Yaskawa INFORM job: R1_W27-A5(90,0)OK-KM.JBI

/JOB
//NAME R1_W27-A5(90,0)OK-KM
///FOLDERNAME KRIS-SCIANA
//POS
///NPOS 202,202,0,12,0,0
///TOOL 0
///POSTYPE PULSE
///PULSE
C00000=17399,70332,19465,-6085,71765,84469
C00001=-37728,-26470,-57837,-12171,79874,87707
C00002=-91138,-151926,-106227,-11663,-44198,37632
C00003=-119745,-150224,-99473,-11370,-45552,35827
C00004=-119745,-150224,-99473,27647,23434,35827
C00005=-82911,-32219,-20746,39404,39160,51491
C00006=-76873,-22201,-13846,34402,37292,54508
C00007=-77767,-15549,-470,39111,33772,51878
C00008=-77963,-13883,2721,40331,32997,51211
C00009=-77963,-13524,3630,40708,32708,51011
C00010=-77963,-13883,2721,40331,32997,51211
C00011=-74912,-26998,-14766,34305,34919,54616
C00012=-87425,-26616,-10195,45168,38615,47962
C00013=-86506,-23763,-6209,45546,37441,47802
C00014=-85850,-22824,-4885,45481,36871,47882
C00015=-86506,-23763,-6209,45546,37441,47802
C00016=-88499,-28370,-15308,43879,40777,48661
C00017=-84065,-38855,-25026,49333,30926,46354
C00018=-97660,-56634,-43247,77155,50749,43385
C00019=-97660,-56634,-43247,77155,50749,-23479
C00020=-84258,-2041,-18253,34253,81408,-37843
C00021=-71650,45427,35116,30336,65668,-37926
C00022=-68559,52359,37552,21834,71082,-35585
C00023=-68559,52806,39758,21974,70033,-35786
C00024=-71650,45427,35116,30336,65668,-37926
C00025=-70945,44875,34529,30103,65482,-37681
C00026=-71650,45427,35116,30336,65668,-37926
C00027=-73638,27357,13179,30116,70049,-37523
C00028=-84818,-6426,-32553,25443,106560,-66628
C00029=-82304,-18386,-36135,24935,102238,-66641
C00030=-82304,-18454,-35234,24871,101700,-66756
C00031=-82304,-18386,-36135,24935,102238,-66641
C00032=-81928,-19848,-37209,24925,102044,-66542
C00033=-82304,-18386,-36135,24935,102238,-66641
C00034=-89590,-10771,-36844,25462,108330,-68030
C00035=-79821,25001,-10397,14026,108535,51508
C00036=-75346,31907,-3594,13981,107184,52914
C00037=-69367,42190,15961,2624,107533,53589
C00038=-69672,41458,15193,2593,107639,53485
C00039=-69367,42204,15728,2627,107683,53592
C00040=-69778,41287,13778,2594,108424,53461
C00041=-69778,41233,14455,2587,107981,53452
C00042=-69778,41399,12679,2608,109158,53478
C00043=-75546,31218,-6024,2098,115588,51477
C00044=-89590,-10931,-36200,25384,107896,-68129
C00045=-81318,-17186,-40796,25354,105117,-65637
C00046=-81011,-18361,-41666,25340,104964,-65554
C00047=-81318,-17186,-40796,25354,105117,-65637
C00048=-81318,-16843,-42196,25499,106059,-65424
C00049=-80508,-20067,-43878,25399,105256,-65302
C00050=-80508,-20199,-43312,25343,104878,-65387
C00051=-80508,-20067,-43878,25399,105256,-65302
C00052=-95846,-36703,-51984,36140,101059,-70811
C00053=-102769,-66525,-54062,50542,79902,-82074
C00054=-102006,-66230,-53915,50487,79519,-81882
C00055=-101071,-65850,-53726,50414,79053,-81646
C00056=-102358,-66368,-53984,50514,79697,-81972
C00057=-109446,-45740,-47717,50613,88014,-81159
C00058=-76818,1585,-28485,25537,105673,-88163
C00059=-74377,-650,-29244,25352,104344,-87556
C00060=-73964,-576,-29181,25336,104222,-87428
C00061=-74377,-650,-29244,25352,104344,-87556
C00062=-74377,-197,-30716,25505,105375,-87324
C00063=-73295,556,-29557,25411,104765,-87062
C00064=-73295,319,-28784,25333,104224,-87184
C00065=-73295,556,-29557,25411,104765,-87062
C00066=-75164,936,-29240,25491,105307,-87630
C00067=-75164,673,-28375,25400,104701,-87767
C00068=-73992,-54,-28979,25351,104361,-87410
C00069=-74218,1135,-29725,25504,105397,-87259
C00070=-70279,39917,7631,24946,101471,-86677
C00071=-70279,39773,8340,24894,101006,-86779
C00072=-70279,39917,7631,24946,101471,-86677
C00073=-71244,40896,8655,24982,101636,-86998
C00074=-70901,41500,10265,24911,100916,-87026
C00075=-70430,41573,10341,24887,100771,-86884
C00076=-70902,41494,10304,24893,100890,-87032
C00077=-61413,47913,18827,22376,82611,-84527
C00078=-60983,48200,19135,22272,82457,-84404
C00079=-61413,47913,18827,22376,82611,-84527
C00080=-61413,48031,17812,22351,83248,-84408
C00081=-60688,48267,18121,22175,82995,-84198
C00082=-60688,48184,18825,22194,82554,-84280
C00083=-60688,48216,18544,22185,82728,-84248
C00084=-61554,48611,18972,22401,82900,-84527
C00085=-61554,48574,19313,22409,82686,-84566
C00086=-61046,48574,19311,22284,82551,-84409
C00087=-61144,49040,18429,22280,83303,-84304
C00088=-63518,19819,-3959,31003,65918,-85445
C00089=-64098,13990,-8483,32812,62419,-85700
C00090=-68885,5858,-4837,49954,39982,-79267
C00091=-65088,14401,2351,47338,37926,-77932
C00092=-64176,16514,4289,46758,37375,-77645
C00093=-64374,16048,3860,46884,37498,-77706
C00094=-64374,16332,5960,47994,36717,-78332
C00095=-65291,19511,8504,48605,37238,-78641
C00096=-67140,20670,8164,49136,38778,-78870
C00097=-66295,22610,10004,48674,38233,-78640
C00098=-66438,22276,9687,48752,38326,-78678
C00099=-66438,22593,11839,49879,37554,-79321
C00100=-66183,17456,6587,49121,37801,-78900
C00101=-69997,303,-8544,51199,40225,-79947
C00102=-70090,462,-8411,51396,40399,61925
C00103=-64431,-7994,-19990,55211,47136,55293
C00104=-59732,2731,-7253,54624,43014,55385
C00105=-61112,6047,-4408,55407,43795,54965
C00106=-58127,6230,-5593,41789,36796,53014
C00107=-57063,4244,-3023,44477,29101,47198
C00108=-49270,4507,-14230,7230,38635,77567
C00109=-52170,-21028,-34442,10411,38272,75983
C00110=-53236,-23757,-36400,11576,38221,75401
C00111=-68411,-26721,-55288,29669,69158,-83075
C00112=-64998,-22231,-39429,29595,61484,-83843
C00113=-47332,3156,-26714,14390,83656,-86934
C00114=-13581,-13792,-41839,5505,90345,-85819
C00115=-16349,-25840,-50577,5581,88837,-86870
C00116=-22627,-48080,-64721,6235,84990,-89226
C00117=-44284,-42364,-63168,13491,82223,-86082
C00118=-48658,384,-30330,14766,84654,-87257
C00119=-13581,-13639,-42286,5505,90698,-85803
C00120=-13581,-13792,-41839,5505,90345,-85819
C00121=-42831,1170,-27974,7852,83268,-89098
C00122=-45008,27799,-716,8149,72970,-89221
C00123=-49813,9029,-19459,14067,72438,-89467
C00124=-51221,-59792,-71163,13641,70093,-81113
C00125=-20731,-35064,-57255,13295,95296,-88132
C00126=-10350,-61458,-73206,13150,96697,-81231
C00127=-18568,-72839,-84924,10276,90748,-67361
C00128=-26792,-78269,-88347,11582,91154,33243
C00129=-45042,-56045,-41152,29344,86284,26690
C00130=-29931,-96865,-59275,30269,72400,28931
C00131=-11330,-93733,-53223,18734,61624,35066
C00132=-13142,-100438,-49115,27852,43711,29575
C00133=-45210,-99902,-50498,43944,62722,17519
C00134=-65059,-105763,-56440,35236,62434,-70425
C00135=-52273,-68840,-35855,24782,78790,-57994
C00136=-44191,-94324,-39451,26680,66575,-57785
C00137=-27622,-61862,-26687,25544,69625,-50822
C00138=-34229,-65282,-33006,25339,73525,-52443
C00139=-29998,-45056,-20412,5383,50998,-19853
C00140=-26959,-13487,10958,4231,47743,-18704
C00141=-30725,7190,27774,5945,48250,-20332
C00142=-26399,12630,34412,-7054,43656,-17025
C00143=-25910,12791,35044,-8483,42971,-16590
C00144=-25523,14356,36662,-10737,43316,-14707
C00145=-25240,1993,23649,-9803,41847,-14580
C00146=-22231,-26812,-1283,-11497,42767,-13220
C00147=-78144,-22833,-14293,20182,52194,33247
C00148=-71297,46898,32867,2677,100084,44239
C00149=-55011,25089,17646,-3023,105619,49711
C00150=-60812,41513,34008,-4227,103729,47709
C00151=-58235,32548,20742,-3759,107403,48505
C00152=-79593,-22722,-23344,19568,57852,33734
C00153=-78528,-18616,-11242,20296,52560,33151
C00154=-78932,-16743,-10167,20417,52946,33052
C00155=-78544,-16737,-8595,20480,51941,33014
C00156=-77955,-18452,-11115,20012,52425,33380
C00157=-78575,-16130,-9486,20269,52757,33170
C00158=-76564,-15411,-8500,18566,50879,33728
C00159=-75844,-13833,-7410,18312,50740,34021
C00160=-76952,-15561,-8970,19469,52340,33810
C00161=-76532,-19770,-12086,19320,52008,33932
C00162=-90733,-10813,-5342,38854,64320,29793
C00163=-90042,-7330,-2603,38655,64092,30029
C00164=-89654,-5763,-1731,38480,64131,30226
C00165=-90645,-6898,-2268,38798,64375,29857
C00166=-90264,-6063,-535,38894,63701,29768
C00167=-89843,-4938,-962,38544,64174,30154
C00168=-90707,-2014,1381,38736,64612,29923
C00169=-91454,1636,4460,38922,64932,29697
C00170=-91128,-2551,1262,38897,64640,29735
C00171=-91822,-6037,-1569,39075,64914,29517
C00172=-89351,12292,-5617,20131,79037,-60764
C00173=-89352,16382,17787,21350,67492,-62811
C00174=-87694,16715,18095,20947,67047,-62250
C00175=-87033,16875,18243,20783,66871,-62026
C00176=-87546,18694,19932,20926,66903,-62219
C00177=-87127,16733,16861,20697,67624,-61924
C00178=-86853,17243,18585,20744,66809,-61967
C00179=-87778,19395,20596,20991,66917,-62307
C00180=-93870,634,-11523,21410,77965,-27109
C00181=-93832,30424,31287,31485,89224,4964
C00182=-93834,30423,31286,31485,89224,4963
C00183=-93835,30423,31286,31485,89225,4963
C00184=-93885,30318,29928,31492,89915,5134
C00185=-93558,28166,29049,31504,89308,5095
C00186=-93835,30423,31286,31484,89222,4963
C00187=-93835,30427,31290,31485,89224,4963
C00188=-93832,30428,31291,31485,89223,4964
C00189=-78422,20921,22036,838,76825,-9185
C00190=-78437,23453,23148,839,77442,-9187
C00191=-77317,26936,27718,-2138,78128,-8741
C00192=-79840,22908,23920,1007,76703,-9676
C00193=-79114,23558,23278,919,77424,-9420
C00194=-78338,20084,11776,-759,84531,-8094
C00195=-114533,-1197,-11881,12870,92966,-10222
C00196=-113047,-131988,-107371,12889,-13343,-10200
C00197=-113047,-158564,-125305,12889,-13343,-10200
C00198=-3699,-158564,-125305,12889,-13343,-10200
C00199=-3699,-158564,-125305,12889,-13343,84424
C00200=5596,-96113,-95019,6240,14020,80272
C00201=27937,63061,-18481,-9952,82568,70189
BC00000=125260,593,1075157
BC00001=243897,593,1075157
BC00002=327653,226,1064237
BC00003=25053,15,1057951
BC00004=25053,15,257506
BC00005=15,15,308848
BC00006=15,15,287123
BC00007=15,15,287123
BC00008=15,15,287123
BC00009=15,15,287123
BC00010=15,15,287123
BC00011=15,15,287123
BC00012=15,15,287123
BC00013=15,15,287123
BC00014=15,15,287123
BC00015=15,15,287123
BC00016=15,15,287123
BC00017=15,15,248984
BC00018=15,15,206829
BC00019=15,15,206829
BC00020=15,15,206829
BC00021=15,15,206829
BC00022=15,15,206829
BC00023=15,15,206829
BC00024=15,15,206829
BC00025=15,15,206826
BC00026=15,15,206829
BC00027=15,15,206829
BC00028=15,15,206829
BC00029=15,15,206829
BC00030=15,15,206829
BC00031=15,15,206829
BC00032=15,15,206829
BC00033=15,15,206829
BC00034=15,15,206829
BC00035=15,15,206829
BC00036=15,15,206829
BC00037=15,15,206829
BC00038=15,15,206829
BC00039=15,15,206829
BC00040=15,15,206829
BC00041=15,15,206829
BC00042=15,15,206829
BC00043=15,15,207086
BC00044=15,15,604261
BC00045=15,15,604261
BC00046=15,15,604261
BC00047=15,15,604261
BC00048=15,15,604261
BC00049=15,15,604261
BC00050=15,15,604261
BC00051=15,15,604261
BC00052=15,15,604261
BC00053=15,15,604261
BC00054=15,15,604261
BC00055=15,15,604261
BC00056=15,15,604261
BC00057=15,15,604261
BC00058=15,15,604261
BC00059=15,15,604261
BC00060=15,15,604261
BC00061=15,15,604261
BC00062=15,15,604261
BC00063=15,15,604261
BC00064=15,15,604261
BC00065=15,15,604261
BC00066=15,15,604261
BC00067=15,15,604261
BC00068=15,15,604261
BC00069=15,15,604261
BC00070=15,15,604261
BC00071=15,15,604261
BC00072=15,15,604261
BC00073=15,15,604261
BC00074=15,15,604259
BC00075=15,15,604259
BC00076=15,15,604261
BC00077=15,32526,604261
BC00078=15,32526,604261
BC00079=15,32526,604261
BC00080=15,32526,604261
BC00081=15,32526,604261
BC00082=15,32526,604261
BC00083=15,32526,604261
BC00084=15,32526,604261
BC00085=15,32526,604261
BC00086=15,32526,604261
BC00087=15,32526,604261
BC00088=15,32526,604261
BC00089=15,32526,604261
BC00090=15,32526,704134
BC00091=15,32526,704134
BC00092=15,32526,704134
BC00093=15,32526,704134
BC00094=17,32524,704134
BC00095=15,32526,704134
BC00096=15,32526,704134
BC00097=15,32526,704134
BC00098=15,32526,704134
BC00099=15,32526,704134
BC00100=15,32526,704134
BC00101=15,32526,704134
BC00102=15,32526,704134
BC00103=15,59931,704134
BC00104=15,59931,704134
BC00105=15,59931,704134
BC00106=15,59931,704134
BC00107=15,59931,704134
BC00108=15,59931,704134
BC00109=15,59931,704134
BC00110=15,59931,704134
BC00111=454,50006,652892
BC00112=454,50006,652892
BC00113=871,66595,604261
BC00114=1930,149815,604260
BC00115=1930,133880,604260
BC00116=1931,106193,604261
BC00117=871,66595,604261
BC00118=871,66595,604261
BC00119=1930,149815,604260
BC00120=1930,149815,604260
BC00121=871,66595,604261
BC00122=871,66595,604261
BC00123=871,66595,604261
BC00124=871,66595,604261
BC00125=871,123107,604261
BC00126=871,123107,604261
BC00127=871,123107,604261
BC00128=871,123107,604261
BC00129=871,123107,812088
BC00130=871,122086,812088
BC00131=871,122086,812088
BC00132=871,122086,812088
BC00133=871,122086,812088
BC00134=871,122086,812088
BC00135=871,122086,424206
BC00136=28253,122086,424206
BC00137=871,122086,424206
BC00138=871,122086,424206
BC00139=871,122086,424206
BC00140=871,122086,424206
BC00141=871,122086,424206
BC00142=871,122086,424206
BC00143=871,122086,424206
BC00144=871,122086,424206
BC00145=871,122086,424206
BC00146=871,122086,424206
BC00147=15,15,317604
BC00148=15,15,317604
BC00149=15,39124,317604
BC00150=15,39124,317604
BC00151=15,39124,317604
BC00152=15,15,296339
BC00153=15,15,296339
BC00154=15,15,287833
BC00155=15,15,287833
BC00156=15,15,287833
BC00157=15,15,287828
BC00158=15,15,287716
BC00159=15,15,287710
BC00160=15,15,296216
BC00161=15,15,317481
BC00162=15,15,307800
BC00163=15,15,285084
BC00164=15,15,275998
BC00165=15,15,275998
BC00166=15,15,275998
BC00167=15,15,276012
BC00168=15,15,276054
BC00169=15,15,276068
BC00170=15,15,285154
BC00171=15,15,307870
BC00172=15,15,362994
BC00173=15,15,362994
BC00174=15,15,341074
BC00175=15,15,332306
BC00176=15,15,332306
BC00177=15,15,332306
BC00178=15,15,332291
BC00179=15,15,362861
BC00180=15,15,362861
BC00181=5357,11188,357193
BC00182=9287,12237,334101
BC00183=10859,12656,324864
BC00184=10859,12656,324864
BC00185=10859,12656,324864
BC00186=11496,12650,324850
BC00187=14702,12223,333954
BC00188=10772,11175,357046
BC00189=6961,15,393964
BC00190=9957,15,370830
BC00191=11155,15,361576
BC00192=11155,15,361576
BC00193=11155,15,361576
BC00194=10008,1318,362128
BC00195=16,10032,390072
BC00196=16,10032,1019085
BC00197=16,10032,1019085
BC00198=124614,10032,1019085
BC00199=354065,10032,1019085
BC00200=328429,10171,1032602
BC00201=164707,10510,1065490
///POSTYPE BASE
///RECTAN
///RCONF 0,0,0,0,1,0,0,0,0,0,0,0,0,0,0,0,0,0,0,0,0,0,0,0
P00006=2.006,1.622,-0.565,0.0000,0.0000,0.0000
P00022=2.006,1.622,-0.565,0.0000,0.0000,0.0000
///RCONF 0,0,0,0,0,0,0,0,0,0,0,0,0,0,0,0,0,0,0,0,0,0,0,0
P00023=-2.957,-4.083,2.762,0.0000,0.0000,0.0000
P00024=-1.466,-0.226,-0.419,0.0000,0.0000,0.0000
P00025=3.643,0.007,-2.585,0.0000,0.0000,0.0000
P00026=2.644,0.055,-2.583,0.0000,0.0000,0.0000
P00027=2.278,0.099,-4.210,0.0000,0.0000,0.0000
P00028=-1.778,-0.182,-2.050,0.0000,0.0000,0.0000
P00029=1.749,4.006,-0.261,0.0000,0.0000,0.0000
P00030=-0.014,-0.768,0.131,0.0000,0.0000,0.0000
P00035=0.390,-0.027,1.040,0.0000,0.0000,0.0000
P00036=-2.434,0.084,0.197,0.0000,0.0000,0.0000
//INST
///DATE 2025/02/07 10:47
///ATTR SC,RW
///GROUP1 RB1,BS1
NOP
SFTOF
MOVJ C00000 BC00000 VJ=100.00
MOVJ C00001 BC00001 VJ=100.00
MOVJ C00002 BC00002 VJ=100.00
MOVJ C00003 BC00003 VJ=100.00
MOVJ C00004 BC00004 VJ=100.00
MOVL C00005 BC00005 V=166.7
MOVL C00006 BC00006 V=166.7
MOVL C00007 BC00007 V=100.0
MOVL C00008 BC00008 V=60.0
REFP 3 C00009 BC00009
CALL JOB:SEARCH-R1
SET P028 P006
SFTON P028
MOVL C00010 BC00010 V=60.0
MOVL C00011 BC00011 V=133.3
MOVL C00012 BC00012 V=133.3
MOVL C00013 BC00013 V=60.0
REFP 3 C00014 BC00014
CALL JOB:SEARCH-R1
SET P028 P006
SFTON P028
MOVL C00015 BC00015 V=60.0
MOVL C00016 BC00016 V=133.3
MOVL C00017 BC00017 V=166.7
'Path S1011
SFTOF
'Path VIA1114
SFTOF
MOVJ C00018 BC00018 VJ=100.00
MOVJ C00019 BC00019 VJ=100.00
'POMIAR NOWE SPOINY
MOVJ C00020 BC00020 VJ=100.00
MOVJ C00021 BC00021 VJ=15.00
MOVL C00022 BC00022 V=83.3
REFP 3 C00023 BC00023
CALL JOB:SEARCH-R1
SET P022 P006
SFTON P022
MOVL C00024 BC00024 V=60.0
REFP 3 C00025 BC00025
CALL JOB:SEARCH-R1
SET P022 P006
SFTON P022
MOVL C00026 BC00026 V=60.0
SFTOF
MOVL C00027 BC00027 V=83.3
MOVL C00028 BC00028 V=83.3
MOVL C00029 BC00029 V=166.7
REFP 3 C00030 BC00030
CALL JOB:SEARCH-R1
SET P023 P006
SFTON P023
MOVL C00031 BC00031 V=60.0
REFP 3 C00032 BC00032
CALL JOB:SEARCH-R1
SET P023 P006
SFTON P023
MOVL C00033 BC00033 V=60.0
MOVJ C00034 BC00034 VJ=15.00
MOVJ C00035 BC00035 VJ=15.00
SFTOF
MOVJ C00036 BC00036 VJ=15.00
'POPRAWIC POMIAR
MOVJ C00037 BC00037 VJ=15.00
REFP 3 C00038 BC00038
CALL JOB:SEARCH-R1
SET P030 P006
SFTON P030
MOVL C00039 BC00039 V=60.0
MOVL C00040 BC00040 V=166.7
REFP 3 C00041 BC00041
CALL JOB:SEARCH-R1
SET P030 P006
SFTON P030
MOVL C00042 BC00042 V=100.0
MOVJ C00043 BC00043 VJ=15.00
SFTOF
MOVJ C00044 BC00044 VJ=50.00
MOVJ C00045 BC00045 VJ=15.00
REFP 3 C00046 BC00046
CALL JOB:SEARCH-R1
SET P024 P006
SFTON P024
MOVL C00047 BC00047 V=60.0
MOVL C00048 BC00048 V=166.7
MOVL C00049 BC00049 V=166.7
REFP 3 C00050 BC00050
CALL JOB:SEARCH-R1
SET P024 P006
SFTON P024
MOVL C00051 BC00051 V=60.0
MOVJ C00052 BC00052 VJ=15.00
SFTOF
MOVJ C00053 BC00053 VJ=15.00
MOVL C00054 BC00054 V=83.3
REFP 3 C00055 BC00055
CALL JOB:SEARCH-R1
SET P025 P006
SFTON P025
MOVL C00056 BC00056 V=83.3
MOVL C00057 BC00057 V=833.3
MOVJ C00058 BC00058 VJ=15.00
MOVL C00059 BC00059 V=100.0
REFP 3 C00060 BC00060
CALL JOB:SEARCH-R1
SET P025 P006
SFTON P025
MOVL C00061 BC00061 V=100.0
MOVL C00062 BC00062 V=166.7
MOVL C00063 BC00063 V=166.7
REFP 3 C00064 BC00064
CALL JOB:SEARCH-R1
SET P025 P006
SFTON P025
MOVL C00065 BC00065 V=166.7
MOVL C00066 BC00066 V=166.7
MOVL C00067 BC00067 V=166.7
REFP 3 C00068 BC00068
CALL JOB:SEARCH-R1
SET P025 P006
SFTON P025
MOVL C00069 BC00069 V=60.0
SFTOF
MOVL C00070 BC00070 V=166.7
REFP 3 C00071 BC00071
CALL JOB:SEARCH-R1
SET P026 P006
SFTON P026
MOVL C00072 BC00072 V=60.0
MOVL C00073 BC00073 V=166.7
MOVL C00074 BC00074 V=166.7
REFP 3 C00075 BC00075
CALL JOB:SEARCH-R1
SET P026 P006
SFTON P026
MOVL C00076 BC00076 V=100.0
SFTOF
MOVL C00077 BC00077 V=166.7
REFP 3 C00078 BC00078
CALL JOB:SEARCH-R1
SET P027 P006
SFTON P027
MOVL C00079 BC00079 V=100.0
MOVL C00080 BC00080 V=166.7
MOVL C00081 BC00081 V=166.7
REFP 3 C00082 BC00082
CALL JOB:SEARCH-R1
SET P027 P006
SFTON P027
MOVL C00083 BC00083 V=100.0
MOVL C00084 BC00084 V=166.7
MOVL C00085 BC00085 V=166.7
REFP 3 C00086 BC00086
CALL JOB:SEARCH-R1
SET P027 P006
SFTON P027
MOVL C00087 BC00087 V=100.0
SFTOF
MOVL C00088 BC00088 V=166.7
MOVJ C00089 BC00089 VJ=15.00
MOVJ C00090 BC00090 VJ=30.00
MOVJ C00091 BC00091 VJ=15.00 PL=0
REFP 3 C00092 BC00092
CALL JOB:SEARCH-R1
SET P035 P006
SFTON P035
MOVL C00093 BC00093 V=60.0
REFP 3 C00094 BC00094
CALL JOB:SEARCH-R1
SET P035 P006
SFTON P035
MOVL C00095 BC00095 V=60.0
SFTOF
MOVJ C00096 BC00096 VJ=15.00 PL=0
REFP 3 C00097 BC00097
CALL JOB:SEARCH-R1
SET P036 P006
SFTON P036
MOVL C00098 BC00098 V=60.0
REFP 3 C00099 BC00099
CALL JOB:SEARCH-R1
SET P036 P006
SFTON P036
MOVL C00100 BC00100 V=60.0
SFTOF
CALL JOB:COFNIJ_DRUT
MOVJ C00101 BC00101 VJ=15.00
MOVJ C00102 BC00102 VJ=15.00
MOVL C00103 BC00103 V=50.0
MACRO1 MJ#(0) ARGF7
SFTON P035
MOVL C00104 BC00104 V=50.0
ARCON
MOVL C00105 BC00105 V=7.5
SFTON P036
MOVL C00106 BC00106 V=7.5
MOVL C00107 BC00107 V=7.5
ARCOF
SFTOF
MOVL C00108 BC00108 V=25.0
MOVL C00109 BC00109 V=66.7
MOVJ C00110 BC00110 VJ=15.00
MOVJ C00111 BC00111 VJ=15.00
MOVJ C00112 BC00112 VJ=15.00
MACRO1 MJ#(0) ARGF7
MOVL C00113 BC00113 V=166.7
SFTON P027
MOVL C00114 BC00114 V=166.7 PL=0
ARCON
SFTON P026
MOVL C00115 BC00115 V=11.7
SFTON P025
MOVL C00116 BC00116 V=11.7
ARCOF
SFTOF
MOVJ C00117 BC00117 VJ=15.00
MOVJ C00118 BC00118 VJ=15.00
SFTON P027
MOVL C00119 BC00119 V=166.7 PL=0
MOVL C00120 BC00120 V=166.7 PL=0
COMM MOVJ C00121 BC00121 VJ=15.00
ARCON
MOVL C00122 BC00122 V=11.7
ARCOF
SFTOF
MOVJ C00123 BC00123 VJ=15.00
MOVJ C00124 BC00124 VJ=15.00
SFTON P026
MOVJ C00125 BC00125 VJ=15.00 PL=0
ARCON
SFTON P025
MOVL C00126 BC00126 V=11.7
ARCOF
SFTOF
MOVJ C00127 BC00127 VJ=15.00
MOVJ C00128 BC00128 VJ=15.00
MOVJ C00129 BC00129 VJ=15.00
MACRO1 MJ#(0) ARGF12
MOVJ C00130 BC00130 VJ=15.00
SFTON P024
MOVJ C00131 BC00131 VJ=15.00
ARCON
MOVL C00132 BC00132 V=12.5
ARCOF
SFTOF
MOVJ C00133 BC00133 VJ=15.00
MOVJ C00134 BC00134 VJ=15.00
MACRO1 MJ#(0) ARGF6
MOVJ C00135 BC00135 VJ=15.00
SFTON P023
MOVJ C00136 BC00136 VJ=15.00
ARCON
MOVL C00137 BC00137 V=9.2
ARCOF
MOVJ C00138 BC00138 VJ=15.00
SFTOF
MOVJ C00139 BC00139 VJ=15.00
SFTON P022
MOVJ C00140 BC00140 VJ=15.00
ARCON
MOVL C00141 BC00141 V=7.5
MOVL C00142 BC00142 V=7.5
MOVL C00143 BC00143 V=7.5
MOVL C00144 BC00144 V=7.5
ARCOF
SFTOF
MOVJ C00145 BC00145 VJ=15.00
MOVJ C00146 BC00146 VJ=15.00
MOVL C00147 BC00147 V=166.7
MACRO1 MJ#(0) ARGF6
MOVL C00148 BC00148 V=83.3
SFTON P030
'POPRAWIC POMIAR
MOVL C00149 BC00149 V=83.3
ARCON
MOVL C00150 BC00150 V=7.5
ARCOF
SFTOF
MOVJ C00151 BC00151 VJ=15.00
COMM MACRO1 MJ#(0) ARGF7
COMM MOVL C00152 BC00152 V=166.7
COMM MOVL C00153 BC00153 V=166.7
COMM SFTON P028
COMM MOVL C00154 BC00154 V=100.0 PL=0
COMM REFP 1 C00155 BC00155
COMM REFP 2 C00156 BC00156
COMM MACRO1 MJ#(0) ARGF7
COMM MOVL C00157 BC00157 V=10.0
COMM MOVL C00158 BC00158 V=10.0
COMM MOVL C00159 BC00159 V=10.0
COMM ARCOF
COMM MOVL C00160 BC00160 V=166.7
COMM MOVL C00161 BC00161 V=166.7
COMM SFTOF
COMM 'Path W1013
COMM SFTOF
COMM SFTON P028
COMM MOVL C00162 BC00162 V=166.7
COMM MOVL C00163 BC00163 V=166.7
COMM MOVL C00164 BC00164 V=100.0 PL=0
COMM REFP 1 C00165 BC00165
COMM REFP 2 C00166 BC00166
COMM MACRO1 MJ#(0) ARGF7
COMM MOVL C00167 BC00167 V=10.0
COMM MOVL C00168 BC00168 V=10.0
COMM MOVL C00169 BC00169 V=10.0
COMM ARCOF
COMM MOVL C00170 BC00170 V=166.7
COMM MOVL C00171 BC00171 V=166.7
COMM SFTOF
COMM 'Path VIA1116
COMM SFTOF
COMM MOVJ C00172 BC00172 VJ=100.00
COMM 'Path W1014
COMM SFTOF
COMM SFTON P028
COMM MOVL C00173 BC00173 V=166.7
COMM MOVL C00174 BC00174 V=166.7
COMM 'NIE SPAWAMY-BRAK MIEJSCA
COMM MOVL C00175 BC00175 V=100.0 PL=0
COMM REFP 1 C00176 BC00176
COMM REFP 2 C00177 BC00177
COMM MACRO1 MJ#(0) ARGF7
COMM MOVL C00178 BC00178 V=10.0
COMM ARCOF
COMM MOVL C00179 BC00179 V=166.7
COMM SFTOF
COMM 'Path VIA1117
COMM SFTOF
COMM MOVJ C00180 BC00180 VJ=100.00
COMM 'Path W1015
COMM SFTOF
COMM SFTON P029
COMM MOVL C00181 BC00181 V=1000.0
COMM MOVL C00182 BC00182 V=400.0
COMM MOVL C00183 BC00183 V=100.0 PL=0
COMM REFP 1 C00184 BC00184
COMM REFP 2 C00185 BC00185
COMM MACRO1 MJ#(0) ARGF0
COMM MOVL C00186 BC00186 V=10.0
COMM ARCOF
COMM MOVL C00187 BC00187 V=400.0
COMM MOVL C00188 BC00188 V=166.7
COMM SFTOF
COMM 'Path W1016
COMM SFTOF
COMM SFTON P029
COMM MOVL C00189 BC00189 V=166.7
COMM MOVL C00190 BC00190 V=166.7
COMM MOVL C00191 BC00191 V=100.0 PL=0
COMM REFP 1 C00192 BC00192
COMM REFP 2 C00193 BC00193
COMM MACRO1 MJ#(0) ARGF7
COMM ARCOF
MOVL C00194 BC00194 V=166.7
SFTOF
MOVJ C00195 BC00195 VJ=100.00
MOVJ C00196 BC00196 VJ=100.00
MOVJ C00197 BC00197 VJ=100.00
MOVJ C00198 BC00198 VJ=100.00
MOVJ C00199 BC00199 VJ=100.00
MOVJ C00200 BC00200 VJ=100.00
MOVJ C00201 BC00201 VJ=40.00
END
